INTERFACE I_MyComponent EXTENDS I_BaseFB

METHOD MyCommand1 : BOOL
VAR_INPUT
END_VAR
END_METHOD

METHOD MyCommand2 : BOOL
VAR_INPUT
END_VAR
END_METHOD

PROPERTY MyVarProperty1 : BOOL
GET
END_GET
SET
END_SET
END_PROPERTY

PROPERTY MyVarProperty2 : BOOL
GET
END_GET
SET
END_SET
END_PROPERTY

END_INTERFACE

(* stored: Version 1.1.0.1, ProductVersion 3.1.4024.12
   Itf I_MyComponent: Id {5d1c1a42-5124-4f65-bcb2-9a123c8b6a66}
   Method MyCommand1: Id {8d94ca5c-baad-4cb7-812f-85deca376178}
   Method MyCommand2: Id {a9de1337-dc5f-4a2b-9b00-889fc1ee2fc9}
   Property MyVarProperty1: Id {1b8ff169-d8a6-4145-bd7c-2bd852f52601}
   Get Get: Id {19c74b8b-da83-45d1-8725-b19e9d9b7f1a}
   Set Set: Id {cb29e313-ebb3-44c6-ac8b-e47b1a7820ba}
   Property MyVarProperty2: Id {9a73445c-ad2b-4470-ae8c-75390a91f31e}
   Get Get: Id {54223792-0e3c-437e-9767-22dbfc43fcc6}
   Set Set: Id {9120bf1c-51b8-448d-98b0-9ae2785cf199} *)
